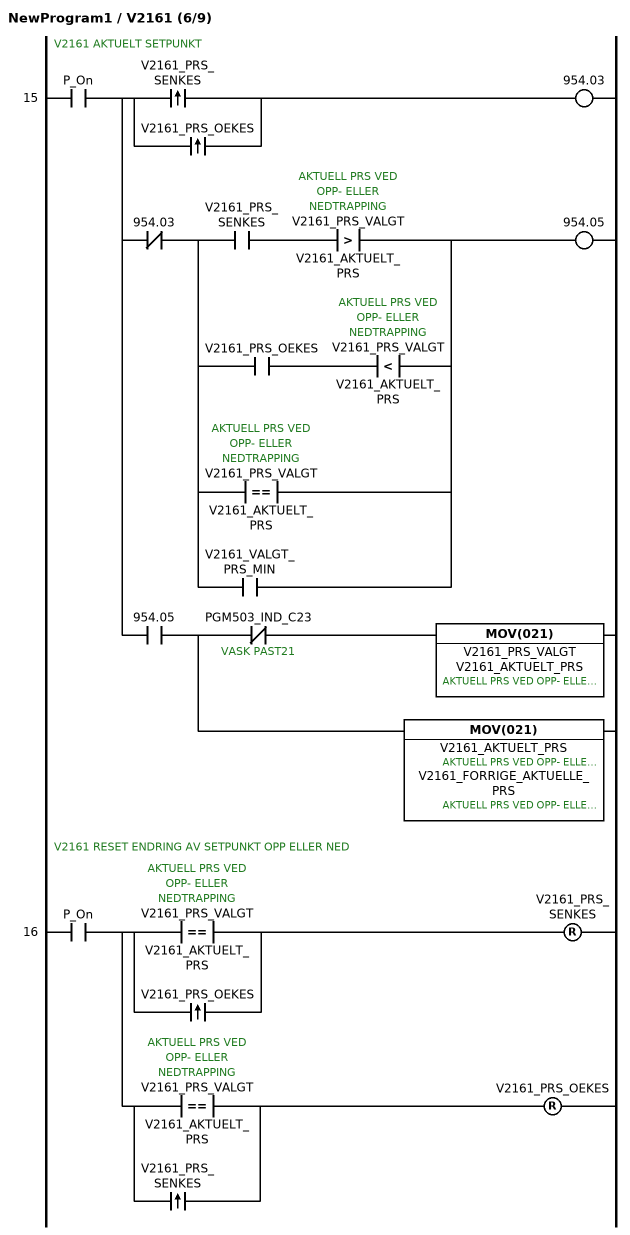
; [picture p1080: NewProgram1 / V2161, rungs 15-16]
; rung 15: V2161 AKTUELT SETPUNKT
LD P_On
OUT TR0
@LD V2161_PRS_SENKES
@OR V2161_PRS_OEKES
ANDLD
OUT 954.03
LD TR0
ANDNOT 954.03
LD V2161_PRS_SENKES
AND>(320) V2161_PRS_VALGT V2161_AKTUELT_PRS  ; AKTUELL PRS VED OPP- ELLER NEDTRAPPING
LD V2161_PRS_OEKES
AND<(310) V2161_PRS_VALGT V2161_AKTUELT_PRS  ; AKTUELL PRS VED OPP- ELLER NEDTRAPPING
ORLD
OR=(300) V2161_PRS_VALGT V2161_AKTUELT_PRS  ; AKTUELL PRS VED OPP- ELLER NEDTRAPPING
OR V2161_VALGT_PRS_MIN
ANDLD
OUT 954.05
LD TR0
AND 954.05
OUT TR0
ANDNOT PGM503_IND_C23  ; VASK PAST21
MOV(021) V2161_PRS_VALGT V2161_AKTUELT_PRS  ; AKTUELL PRS VED OPP- ELLER NEDTRAPPING
LD TR0
MOV(021) V2161_AKTUELT_PRS V2161_FORRIGE_AKTUELLE_PRS  ; AKTUELL PRS VED OPP- ELLER NEDTRAPPING
; rung 16: V2161 RESET ENDRING AV SETPUNKT OPP ELLER NED
LD P_On
OUT TR0
LD=(300) V2161_PRS_VALGT V2161_AKTUELT_PRS  ; AKTUELL PRS VED OPP- ELLER NEDTRAPPING
@OR V2161_PRS_OEKES
ANDLD
RSET V2161_PRS_SENKES
LD TR0
LD=(300) V2161_PRS_VALGT V2161_AKTUELT_PRS  ; AKTUELL PRS VED OPP- ELLER NEDTRAPPING
@OR V2161_PRS_SENKES
ANDLD
RSET V2161_PRS_OEKES

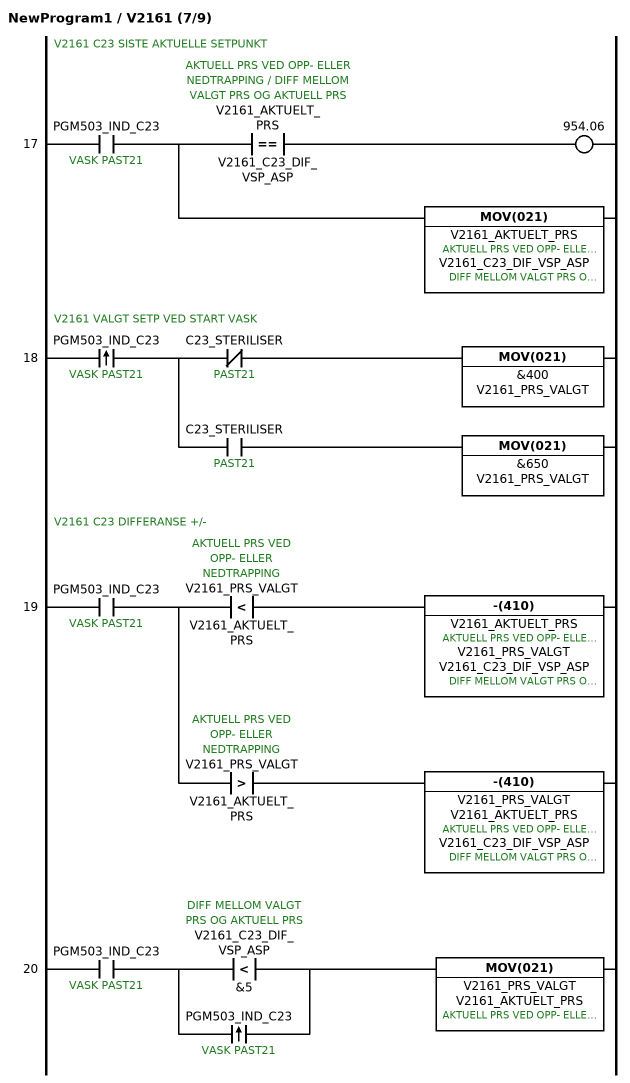
; rung 17: V2161 C23 SISTE AKTUELLE SETPUNKT
LD PGM503_IND_C23  ; VASK PAST21
OUT TR0
AND=(300) V2161_AKTUELT_PRS V2161_C23_DIF_VSP_ASP  ; AKTUELL PRS VED OPP- ELLER NEDTRAPPING, DIFF MELLOM VALGT PRS OG AKTUELL PRS
OUT 954.06
LD TR0
MOV(021) V2161_AKTUELT_PRS V2161_C23_DIF_VSP_ASP  ; AKTUELL PRS VED OPP- ELLER NEDTRAPPING, DIFF MELLOM VALGT PRS OG AKTUELL PRS
; rung 18: V2161 VALGT SETP VED START VASK
@LD PGM503_IND_C23  ; VASK PAST21
OUT TR0
ANDNOT C23_STERILISER  ; PAST21
MOV(021) &400 V2161_PRS_VALGT
LD TR0
AND C23_STERILISER  ; PAST21
MOV(021) &650 V2161_PRS_VALGT
; rung 19: V2161 C23 DIFFERANSE +/-
LD PGM503_IND_C23  ; VASK PAST21
OUT TR0
AND<(310) V2161_PRS_VALGT V2161_AKTUELT_PRS  ; AKTUELL PRS VED OPP- ELLER NEDTRAPPING
-(410) V2161_AKTUELT_PRS V2161_PRS_VALGT V2161_C23_DIF_VSP_ASP  ; AKTUELL PRS VED OPP- ELLER NEDTRAPPING, DIFF MELLOM VALGT PRS OG AKTUELL PRS
LD TR0
AND>(320) V2161_PRS_VALGT V2161_AKTUELT_PRS  ; AKTUELL PRS VED OPP- ELLER NEDTRAPPING
-(410) V2161_PRS_VALGT V2161_AKTUELT_PRS V2161_C23_DIF_VSP_ASP  ; AKTUELL PRS VED OPP- ELLER NEDTRAPPING, DIFF MELLOM VALGT PRS OG AKTUELL PRS
; rung 20
LD PGM503_IND_C23  ; VASK PAST21
LD<(310) V2161_C23_DIF_VSP_ASP &5  ; DIFF MELLOM VALGT PRS OG AKTUELL PRS
@OR PGM503_IND_C23  ; VASK PAST21
ANDLD
MOV(021) V2161_PRS_VALGT V2161_AKTUELT_PRS  ; AKTUELL PRS VED OPP- ELLER NEDTRAPPING

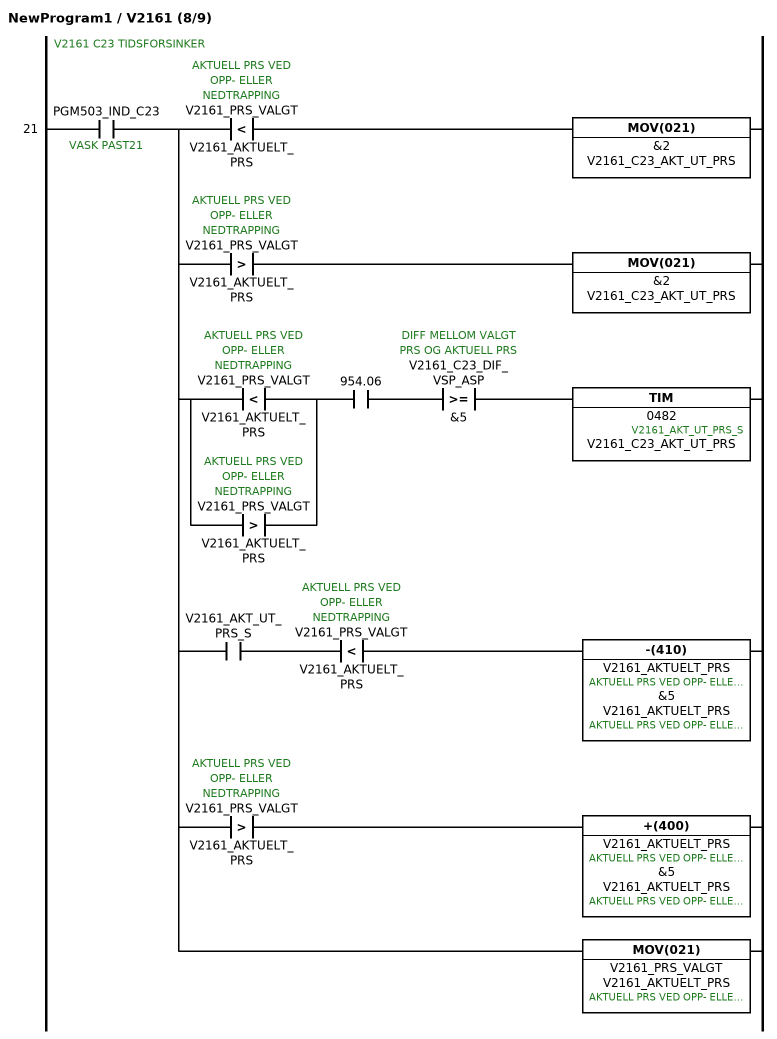
; rung 21: V2161 C23 TIDSFORSINKER
LD PGM503_IND_C23  ; VASK PAST21
OUT TR0
AND<(310) V2161_PRS_VALGT V2161_AKTUELT_PRS  ; AKTUELL PRS VED OPP- ELLER NEDTRAPPING
MOV(021) &2 V2161_C23_AKT_UT_PRS
LD TR0
AND>(320) V2161_PRS_VALGT V2161_AKTUELT_PRS  ; AKTUELL PRS VED OPP- ELLER NEDTRAPPING
MOV(021) &2 V2161_C23_AKT_UT_PRS
LD TR0
LD<(310) V2161_PRS_VALGT V2161_AKTUELT_PRS  ; AKTUELL PRS VED OPP- ELLER NEDTRAPPING
OR>(320) V2161_PRS_VALGT V2161_AKTUELT_PRS  ; AKTUELL PRS VED OPP- ELLER NEDTRAPPING
ANDLD
AND 954.06
AND>=(325) V2161_C23_DIF_VSP_ASP &5  ; DIFF MELLOM VALGT PRS OG AKTUELL PRS
TIM 0482 V2161_C23_AKT_UT_PRS  ; V2161_AKT_UT_PRS_S
LD TR0
AND V2161_AKT_UT_PRS_S
AND<(310) V2161_PRS_VALGT V2161_AKTUELT_PRS  ; AKTUELL PRS VED OPP- ELLER NEDTRAPPING
-(410) V2161_AKTUELT_PRS &5 V2161_AKTUELT_PRS  ; AKTUELL PRS VED OPP- ELLER NEDTRAPPING
LD TR0
AND>(320) V2161_PRS_VALGT V2161_AKTUELT_PRS  ; AKTUELL PRS VED OPP- ELLER NEDTRAPPING
+(400) V2161_AKTUELT_PRS &5 V2161_AKTUELT_PRS  ; AKTUELL PRS VED OPP- ELLER NEDTRAPPING
LD TR0
MOV(021) V2161_PRS_VALGT V2161_AKTUELT_PRS  ; AKTUELL PRS VED OPP- ELLER NEDTRAPPING

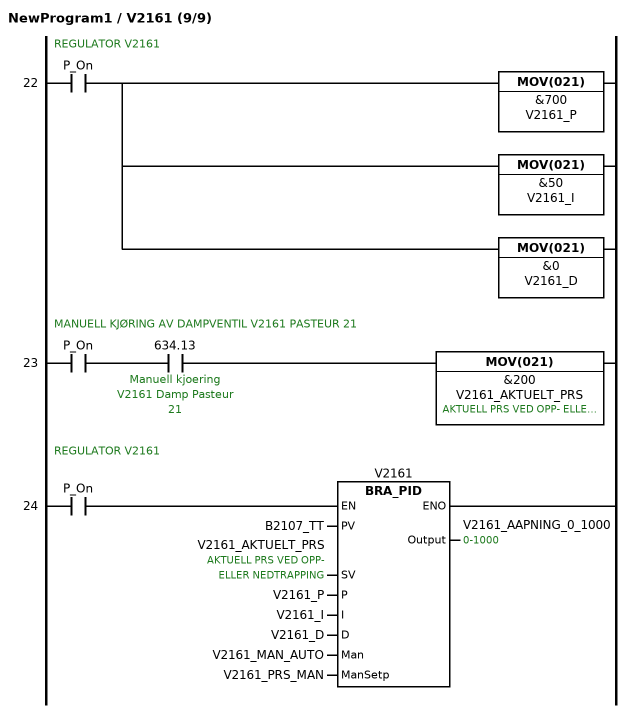
; rung 22: REGULATOR V2161
LD P_On
MOV(021) &700 V2161_P
MOV(021) &50 V2161_I
MOV(021) &0 V2161_D
; rung 23: MANUELL KJØRING AV DAMPVENTIL V2161 PASTEUR 21
LD P_On
AND 634.13  ; Manuell kjoering V2161 Damp Pasteur 21
MOV(021) &200 V2161_AKTUELT_PRS  ; AKTUELL PRS VED OPP- ELLER NEDTRAPPING
; rung 24: REGULATOR V2161
LD P_On
CALL V2161 : BRA_PID (PV := B2107_TT, SV := V2161_AKTUELT_PRS, P := V2161_P, I := V2161_I, D := V2161_D, Man := V2161_MAN_AUTO, ManSetp := V2161_PRS_MAN, Output => V2161_AAPNING_0_1000)  ; AKTUELL PRS VED OPP- ELLER NEDTRAPPING, 0-1000

### Section SEP21_KOMMUNIKASJ0N
; Kriterier: / - Separator går automatisk i "standby" etter "Start Up" / - Hvis ikke flow etter "Start Up", sett separator i "Feed Off" / - Ved skudd tar separator ikke mot nye kommandoer. La kommandoer stå høyt til ferdig. / GJENSTÅR: / - Kryssing av profibuss adresser

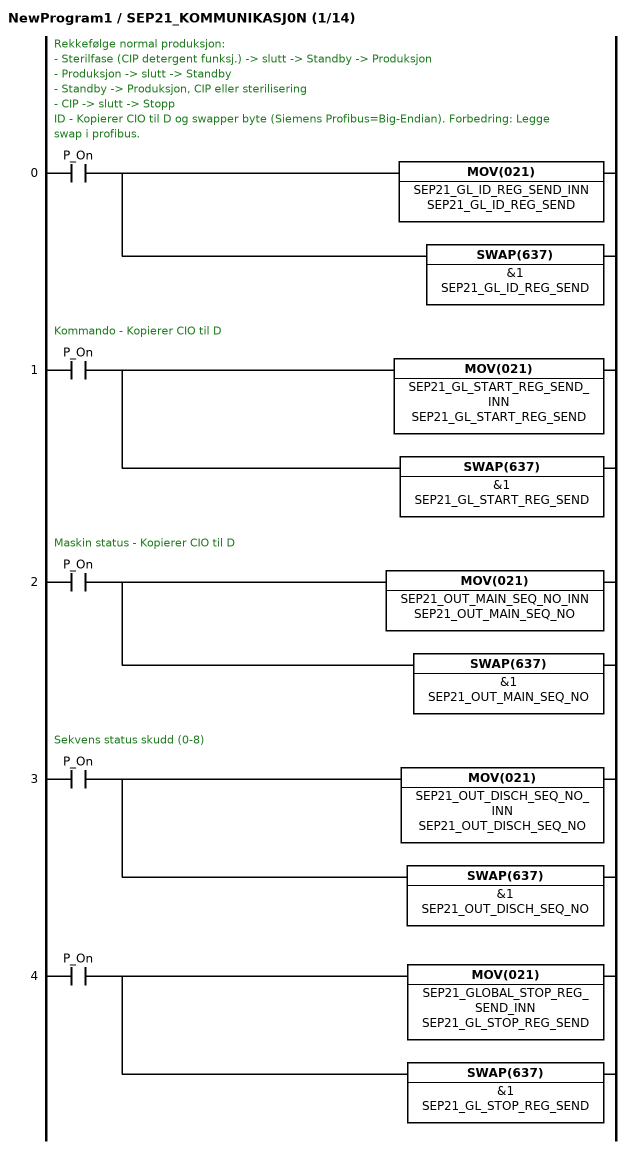
; rung 0: Rekkefølge normal produksjon: / - Sterilfase (CIP detergent funksj.) -> slutt -> Standby -> Produksjon / - Produksjon -> slutt -> Standby / - Standby -> Produksjon, CIP eller sterilisering / - CIP -> slutt -> Stopp / ID - Kopierer CIO til D og swapper byte (Siemens Profibus=Big-Endian). Forbedring: Legge swap i profibus.
LD P_On
MOV(021) SEP21_GL_ID_REG_SEND_INN SEP21_GL_ID_REG_SEND
SWAP(637) &1 SEP21_GL_ID_REG_SEND
; rung 1: Kommando - Kopierer CIO til D
LD P_On
MOV(021) SEP21_GL_START_REG_SEND_INN SEP21_GL_START_REG_SEND
SWAP(637) &1 SEP21_GL_START_REG_SEND
; rung 2: Maskin status - Kopierer CIO til D
LD P_On
MOV(021) SEP21_OUT_MAIN_SEQ_NO_INN SEP21_OUT_MAIN_SEQ_NO
SWAP(637) &1 SEP21_OUT_MAIN_SEQ_NO
; rung 3: Sekvens status skudd (0-8)
LD P_On
MOV(021) SEP21_OUT_DISCH_SEQ_NO_INN SEP21_OUT_DISCH_SEQ_NO
SWAP(637) &1 SEP21_OUT_DISCH_SEQ_NO
; rung 4
LD P_On
MOV(021) SEP21_GLOBAL_STOP_REG_SEND_INN SEP21_GL_STOP_REG_SEND
SWAP(637) &1 SEP21_GL_STOP_REG_SEND

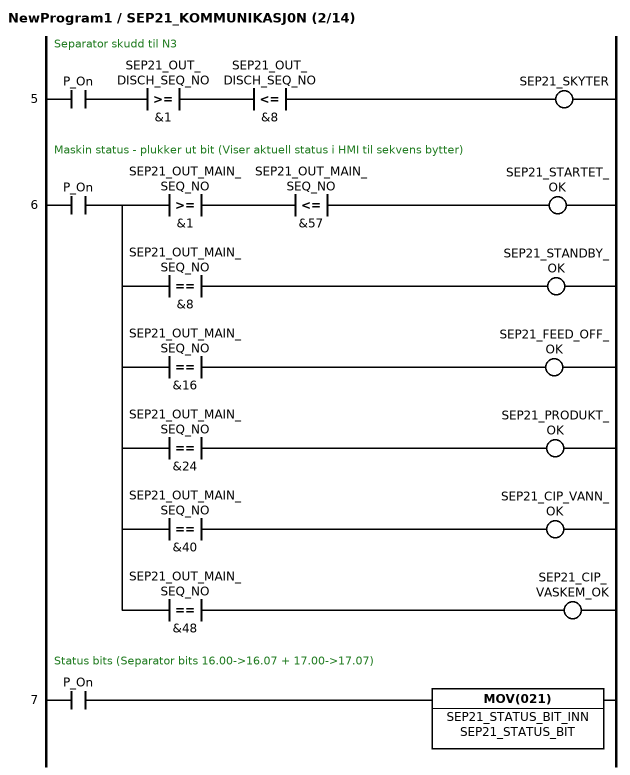
; rung 5: Separator skudd til N3
LD P_On
AND>=(325) SEP21_OUT_DISCH_SEQ_NO &1
AND<=(315) SEP21_OUT_DISCH_SEQ_NO &8
OUT SEP21_SKYTER
; rung 6: Maskin status - plukker ut bit (Viser aktuell status i HMI til sekvens bytter)
LD P_On
OUT TR0
AND>=(325) SEP21_OUT_MAIN_SEQ_NO &1
AND<=(315) SEP21_OUT_MAIN_SEQ_NO &57
OUT SEP21_STARTET_OK
LD TR0
AND=(300) SEP21_OUT_MAIN_SEQ_NO &8
OUT SEP21_STANDBY_OK
LD TR0
AND=(300) SEP21_OUT_MAIN_SEQ_NO &16
OUT SEP21_FEED_OFF_OK
LD TR0
AND=(300) SEP21_OUT_MAIN_SEQ_NO &24
OUT SEP21_PRODUKT_OK
LD TR0
AND=(300) SEP21_OUT_MAIN_SEQ_NO &40
OUT SEP21_CIP_VANN_OK
LD TR0
AND=(300) SEP21_OUT_MAIN_SEQ_NO &48
OUT SEP21_CIP_VASKEM_OK
; rung 7: Status bits (Separator bits 16.00->16.07 + 17.00->17.07)
LD P_On
MOV(021) SEP21_STATUS_BIT_INN SEP21_STATUS_BIT

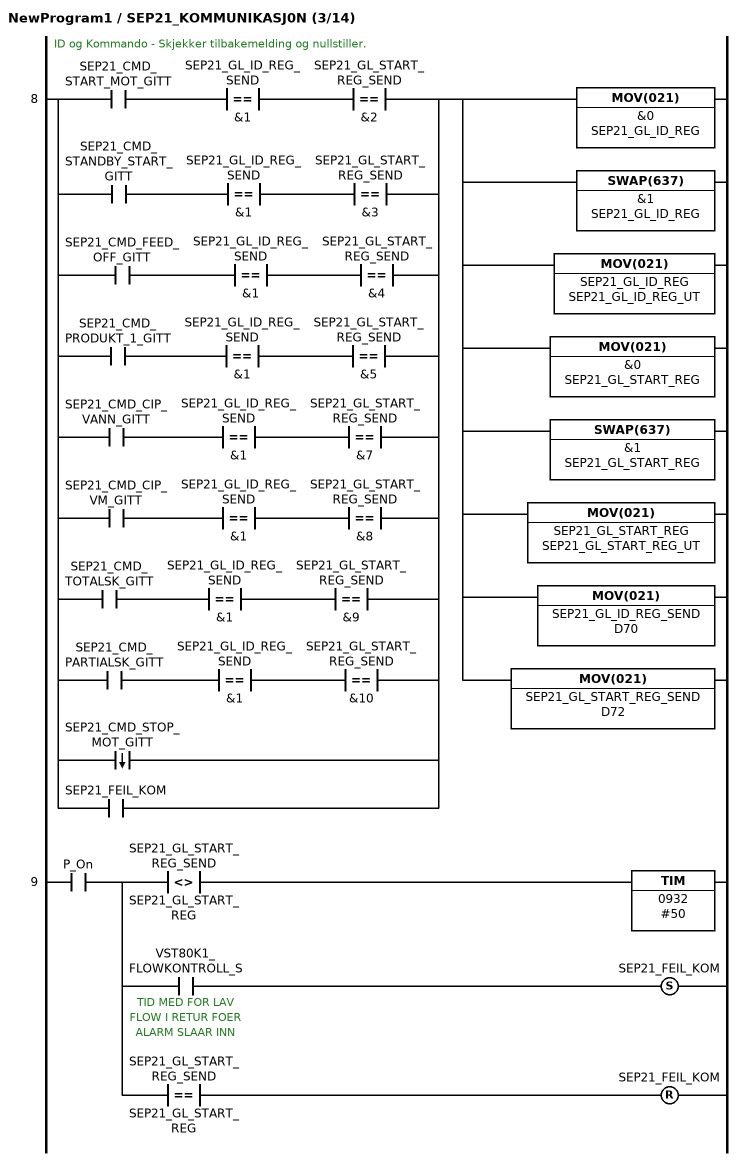
; rung 8: ID og Kommando - Skjekker tilbakemelding og nullstiller.
LD SEP21_CMD_START_MOT_GITT
AND=(300) SEP21_GL_ID_REG_SEND &1
AND=(300) SEP21_GL_START_REG_SEND &2
LD SEP21_CMD_STANDBY_START_GITT
AND=(300) SEP21_GL_ID_REG_SEND &1
AND=(300) SEP21_GL_START_REG_SEND &3
ORLD
LD SEP21_CMD_FEED_OFF_GITT
AND=(300) SEP21_GL_ID_REG_SEND &1
AND=(300) SEP21_GL_START_REG_SEND &4
ORLD
LD SEP21_CMD_PRODUKT_1_GITT
AND=(300) SEP21_GL_ID_REG_SEND &1
AND=(300) SEP21_GL_START_REG_SEND &5
ORLD
LD SEP21_CMD_CIP_VANN_GITT
AND=(300) SEP21_GL_ID_REG_SEND &1
AND=(300) SEP21_GL_START_REG_SEND &7
ORLD
LD SEP21_CMD_CIP_VM_GITT
AND=(300) SEP21_GL_ID_REG_SEND &1
AND=(300) SEP21_GL_START_REG_SEND &8
ORLD
LD SEP21_CMD_TOTALSK_GITT
AND=(300) SEP21_GL_ID_REG_SEND &1
AND=(300) SEP21_GL_START_REG_SEND &9
ORLD
LD SEP21_CMD_PARTIALSK_GITT
AND=(300) SEP21_GL_ID_REG_SEND &1
AND=(300) SEP21_GL_START_REG_SEND &10
ORLD
%OR SEP21_CMD_STOP_MOT_GITT  // Hvis stop så nullstill register
OR SEP21_FEIL_KOM
MOV(021) &0 SEP21_GL_ID_REG
SWAP(637) &1 SEP21_GL_ID_REG
MOV(021) SEP21_GL_ID_REG SEP21_GL_ID_REG_UT
MOV(021) &0 SEP21_GL_START_REG
SWAP(637) &1 SEP21_GL_START_REG
MOV(021) SEP21_GL_START_REG SEP21_GL_START_REG_UT
MOV(021) SEP21_GL_ID_REG_SEND D70  // For test - Siste ID som er mottatt
MOV(021) SEP21_GL_START_REG_SEND D72  // For test - Siste KOMMANDO som er mottatt
; rung 9
LD P_On
OUT TR0
AND<>(305) SEP21_GL_START_REG_SEND SEP21_GL_START_REG
TIM 0932 #50
LD TR0
AND VST80K1_FLOWKONTROLL_S  ; TID MED FOR LAV FLOW I RETUR FOER ALARM SLAAR INN
SET SEP21_FEIL_KOM
LD TR0
AND=(300) SEP21_GL_START_REG_SEND SEP21_GL_START_REG
RSET SEP21_FEIL_KOM

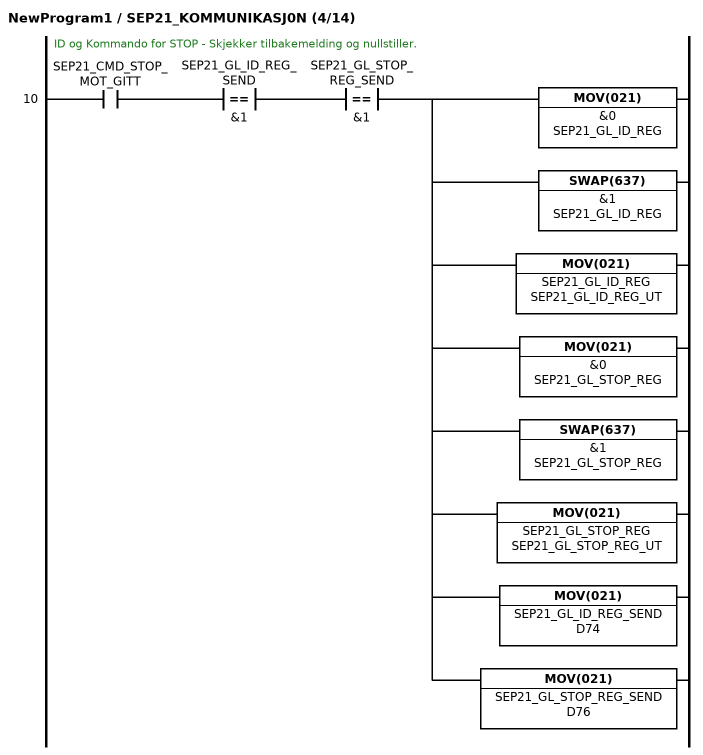
; rung 10: ID og Kommando for STOP - Skjekker tilbakemelding og nullstiller.
LD SEP21_CMD_STOP_MOT_GITT
AND=(300) SEP21_GL_ID_REG_SEND &1
AND=(300) SEP21_GL_STOP_REG_SEND &1
MOV(021) &0 SEP21_GL_ID_REG
SWAP(637) &1 SEP21_GL_ID_REG
MOV(021) SEP21_GL_ID_REG SEP21_GL_ID_REG_UT
MOV(021) &0 SEP21_GL_STOP_REG
SWAP(637) &1 SEP21_GL_STOP_REG
MOV(021) SEP21_GL_STOP_REG SEP21_GL_STOP_REG_UT
MOV(021) SEP21_GL_ID_REG_SEND D74  // For test - Siste STOP ID som er mottatt
MOV(021) SEP21_GL_STOP_REG_SEND D76  // For test - Siste STOP KOMMANDO som er mottatt

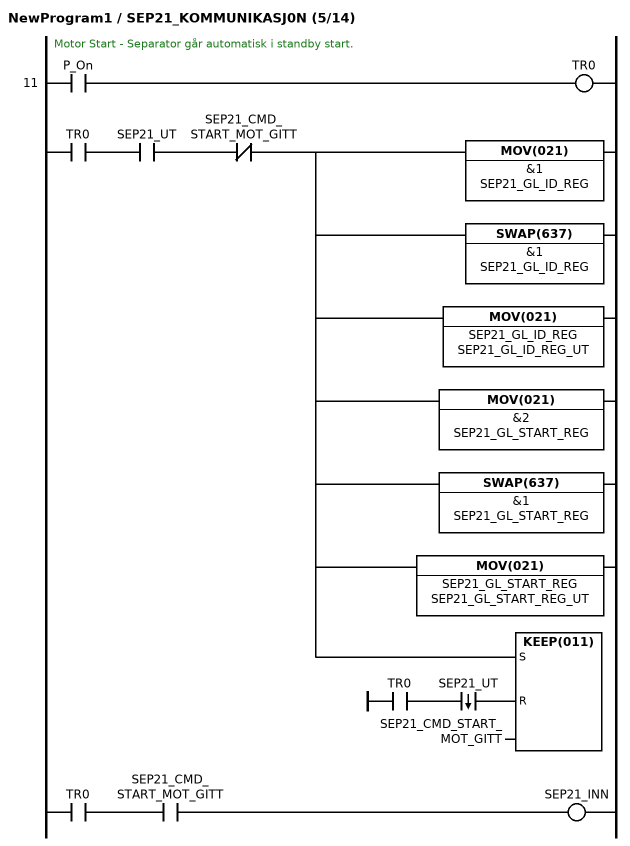
; rung 11: Motor Start - Separator går automatisk i standby start.
LD P_On
OUT TR0
AND SEP21_UT
ANDNOT SEP21_CMD_START_MOT_GITT
MOV(021) &1 SEP21_GL_ID_REG
SWAP(637) &1 SEP21_GL_ID_REG
MOV(021) SEP21_GL_ID_REG SEP21_GL_ID_REG_UT
MOV(021) &2 SEP21_GL_START_REG
SWAP(637) &1 SEP21_GL_START_REG
MOV(021) SEP21_GL_START_REG SEP21_GL_START_REG_UT
LD TR0
%AND SEP21_UT
KEEP(011) SEP21_CMD_START_MOT_GITT
LD TR0
AND SEP21_CMD_START_MOT_GITT
OUT SEP21_INN

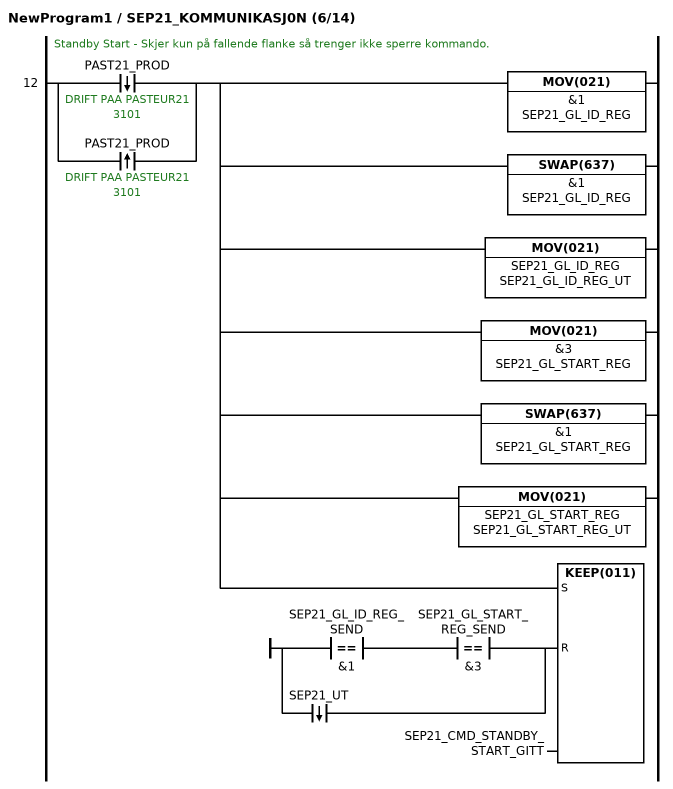
; rung 12: Standby Start - Skjer kun på fallende flanke så trenger ikke sperre kommando.
%LD PAST21_PROD  ; DRIFT PAA PASTEUR21 3101
@OR PAST21_PROD  ; DRIFT PAA PASTEUR21 3101  // Kan ikke gå direkte til prod 1 fra CIP detergent. Må via Standby, stopp eller CIP vann.
MOV(021) &1 SEP21_GL_ID_REG
SWAP(637) &1 SEP21_GL_ID_REG
MOV(021) SEP21_GL_ID_REG SEP21_GL_ID_REG_UT
MOV(021) &3 SEP21_GL_START_REG
SWAP(637) &1 SEP21_GL_START_REG
MOV(021) SEP21_GL_START_REG SEP21_GL_START_REG_UT
LD=(300) SEP21_GL_ID_REG_SEND &1
AND=(300) SEP21_GL_START_REG_SEND &3
%OR SEP21_UT
KEEP(011) SEP21_CMD_STANDBY_START_GITT

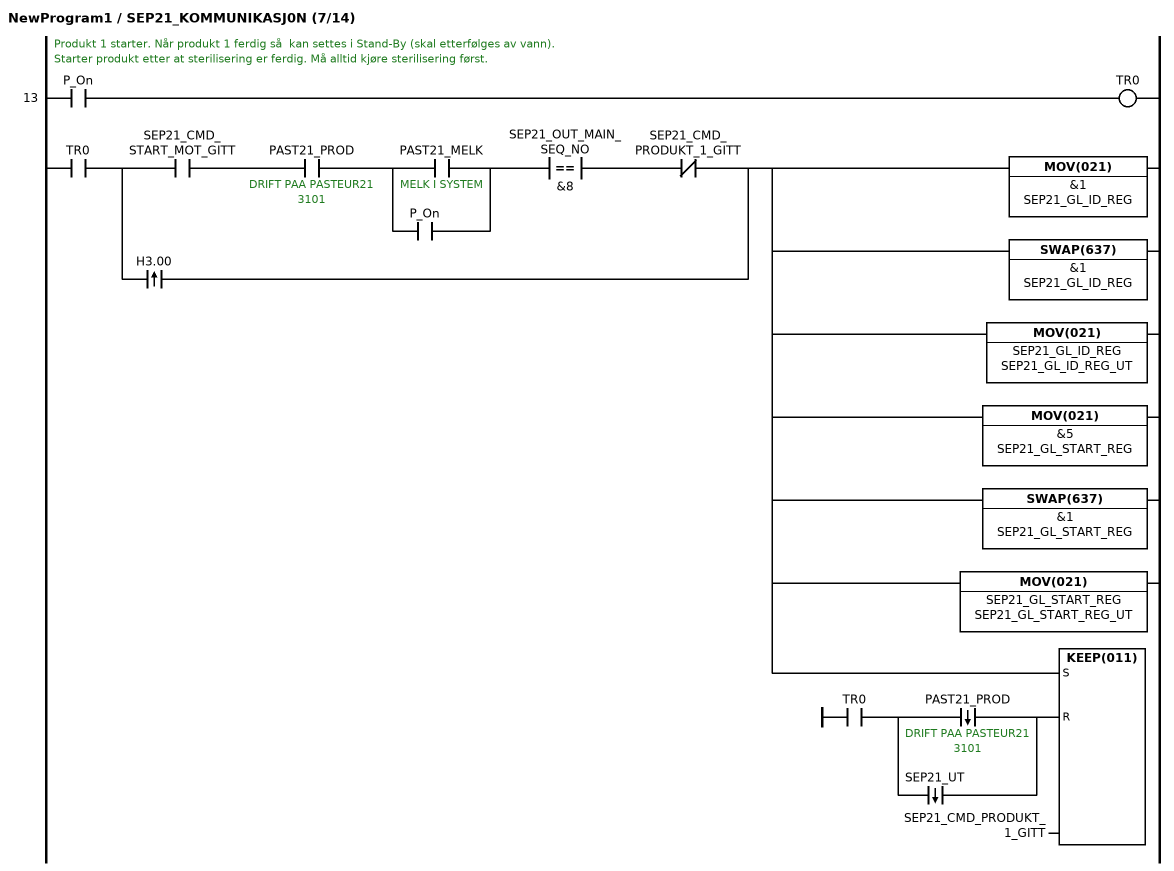
; rung 13: Produkt 1 starter. Når produkt 1 ferdig så  kan settes i Stand-By (skal etterfølges av vann). / Starter produkt etter at sterilisering er ferdig. Må alltid kjøre sterilisering først.
LD P_On
OUT TR0
LD SEP21_CMD_START_MOT_GITT
AND PAST21_PROD  ; DRIFT PAA PASTEUR21 3101
LD PAST21_MELK  ; MELK I SYSTEM
OR P_On
ANDLD
AND=(300) SEP21_OUT_MAIN_SEQ_NO &8  // Kann ikke gå direkte til prod1 fra CIP detergent (se manual). Må via Standby.
ANDNOT SEP21_CMD_PRODUKT_1_GITT
@OR H3.00
ANDLD
MOV(021) &1 SEP21_GL_ID_REG
SWAP(637) &1 SEP21_GL_ID_REG
MOV(021) SEP21_GL_ID_REG SEP21_GL_ID_REG_UT
MOV(021) &5 SEP21_GL_START_REG
SWAP(637) &1 SEP21_GL_START_REG
MOV(021) SEP21_GL_START_REG SEP21_GL_START_REG_UT
LD TR0
%LD PAST21_PROD  ; DRIFT PAA PASTEUR21 3101
%OR SEP21_UT
ANDLD
KEEP(011) SEP21_CMD_PRODUKT_1_GITT

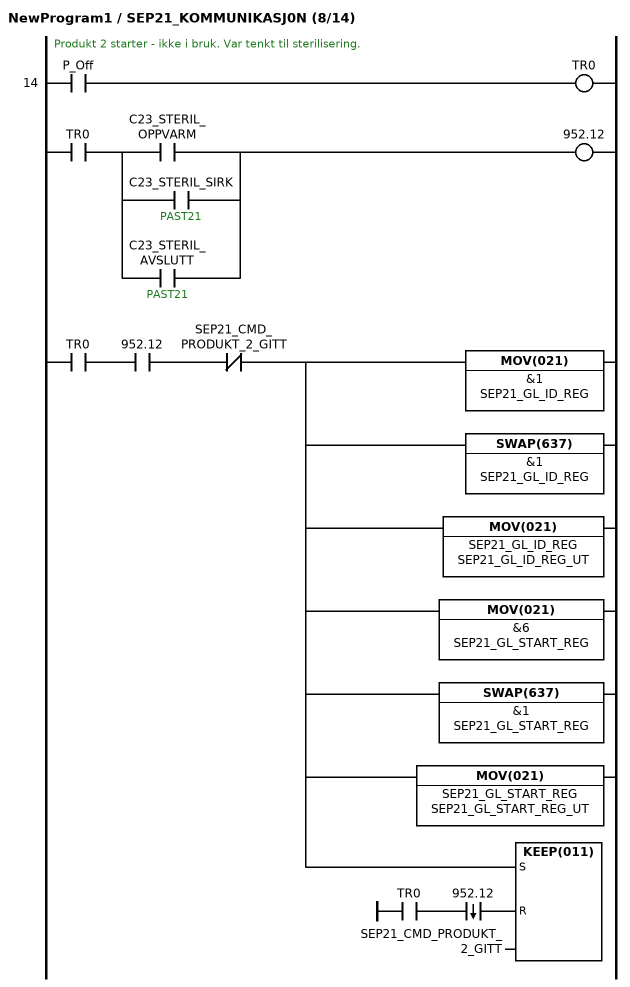
; rung 14: Produkt 2 starter - ikke i bruk. Var tenkt til sterilisering.
LD P_Off
OUT TR0
LD C23_STERIL_OPPVARM
OR C23_STERIL_SIRK  ; PAST21
OR C23_STERIL_AVSLUTT  ; PAST21
ANDLD
OUT 952.12
LD TR0
AND 952.12
ANDNOT SEP21_CMD_PRODUKT_2_GITT
MOV(021) &1 SEP21_GL_ID_REG
SWAP(637) &1 SEP21_GL_ID_REG
MOV(021) SEP21_GL_ID_REG SEP21_GL_ID_REG_UT
MOV(021) &6 SEP21_GL_START_REG
SWAP(637) &1 SEP21_GL_START_REG
MOV(021) SEP21_GL_START_REG SEP21_GL_START_REG_UT
LD TR0
%AND 952.12
KEEP(011) SEP21_CMD_PRODUKT_2_GITT

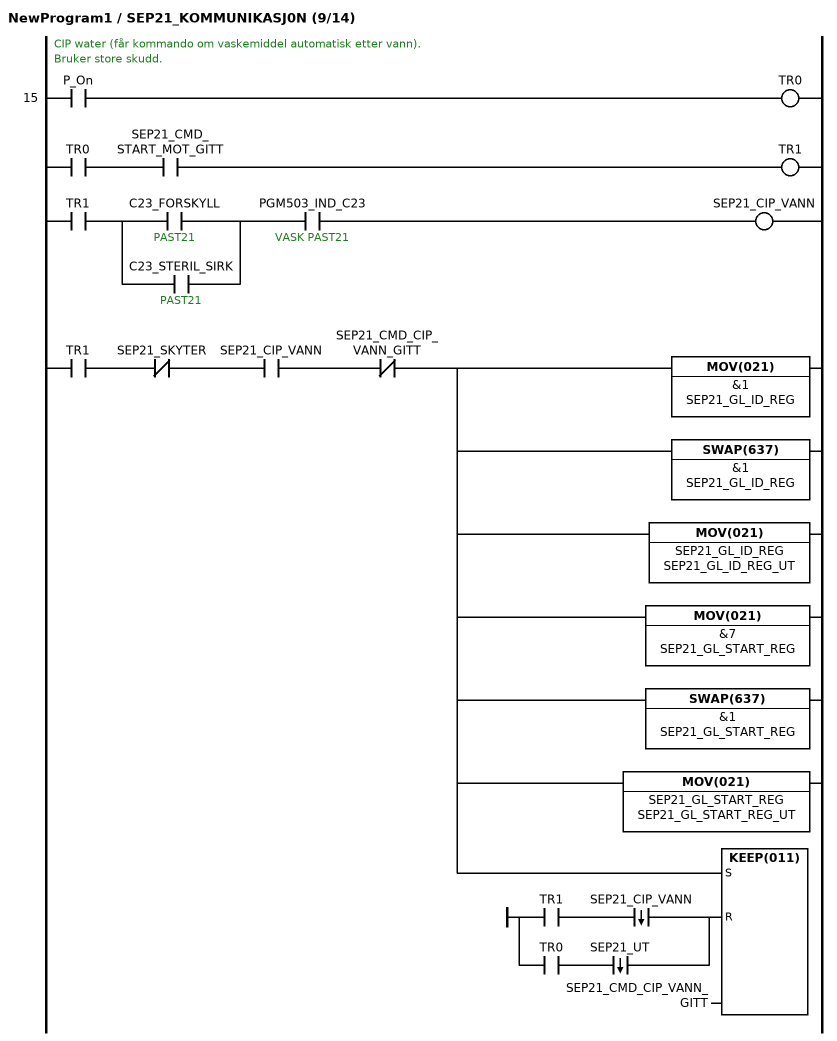
; rung 15: CIP water (får kommando om vaskemiddel automatisk etter vann). / Bruker store skudd.
LD P_On
OUT TR0
AND SEP21_CMD_START_MOT_GITT
OUT TR1
LD C23_FORSKYLL  ; PAST21
OR C23_STERIL_SIRK  ; PAST21
ANDLD
AND PGM503_IND_C23  ; VASK PAST21
OUT SEP21_CIP_VANN
LD TR1
ANDNOT SEP21_SKYTER
AND SEP21_CIP_VANN
ANDNOT SEP21_CMD_CIP_VANN_GITT
MOV(021) &1 SEP21_GL_ID_REG
SWAP(637) &1 SEP21_GL_ID_REG
MOV(021) SEP21_GL_ID_REG SEP21_GL_ID_REG_UT
MOV(021) &7 SEP21_GL_START_REG
SWAP(637) &1 SEP21_GL_START_REG
MOV(021) SEP21_GL_START_REG SEP21_GL_START_REG_UT
LD TR1
%AND SEP21_CIP_VANN
LD TR0
%AND SEP21_UT
ORLD
KEEP(011) SEP21_CMD_CIP_VANN_GITT

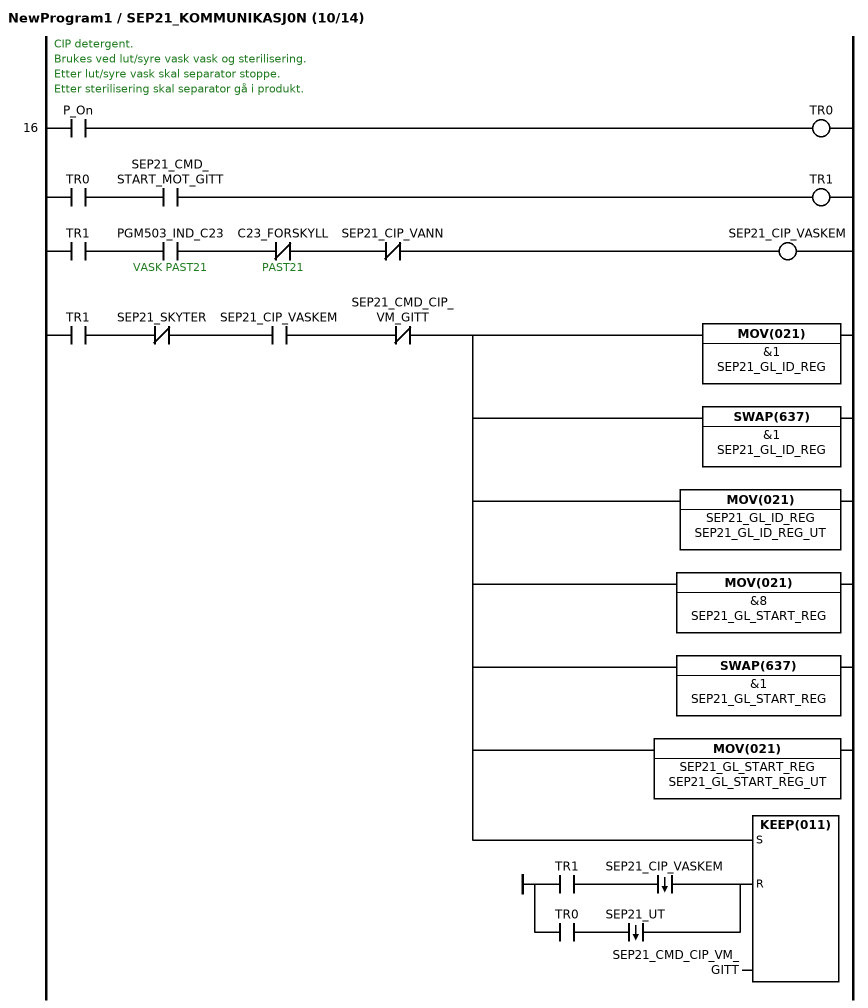
; rung 16: CIP detergent. / Brukes ved lut/syre vask vask og sterilisering. / Etter lut/syre vask skal separator stoppe. / Etter sterilisering skal separator gå i produkt.
LD P_On
OUT TR0
AND SEP21_CMD_START_MOT_GITT
OUT TR1
AND PGM503_IND_C23  ; VASK PAST21
ANDNOT C23_FORSKYLL  ; PAST21
ANDNOT SEP21_CIP_VANN  // Midlertidig. 3616.11 toggler av/på ved start av CIP vann! Må rettes i Node3. / 3616.11 går også på ved sterilvask. Da trenger vi egentlig ikke sterilvask fra ipc så lenge CIP detergant kan brukes som sterilvask.
OUT SEP21_CIP_VASKEM
LD TR1
ANDNOT SEP21_SKYTER
AND SEP21_CIP_VASKEM
ANDNOT SEP21_CMD_CIP_VM_GITT
MOV(021) &1 SEP21_GL_ID_REG
SWAP(637) &1 SEP21_GL_ID_REG
MOV(021) SEP21_GL_ID_REG SEP21_GL_ID_REG_UT
MOV(021) &8 SEP21_GL_START_REG
SWAP(637) &1 SEP21_GL_START_REG
MOV(021) SEP21_GL_START_REG SEP21_GL_START_REG_UT
LD TR1
%AND SEP21_CIP_VASKEM
LD TR0
%AND SEP21_UT
ORLD
KEEP(011) SEP21_CMD_CIP_VM_GITT

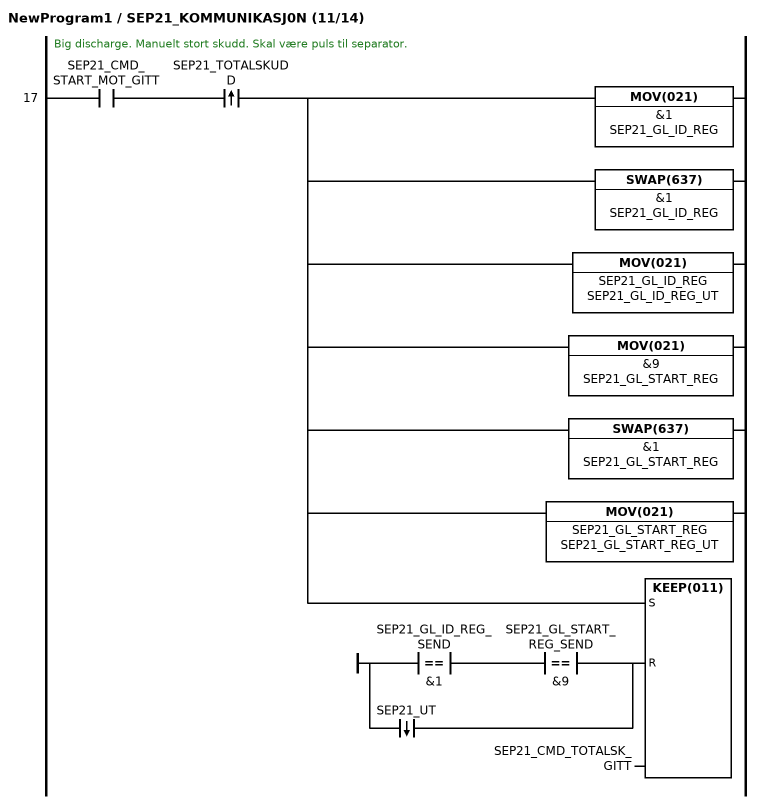
; rung 17: Big discharge. Manuelt stort skudd. Skal være puls til separator.
LD SEP21_CMD_START_MOT_GITT
@AND SEP21_TOTALSKUDD
MOV(021) &1 SEP21_GL_ID_REG
SWAP(637) &1 SEP21_GL_ID_REG
MOV(021) SEP21_GL_ID_REG SEP21_GL_ID_REG_UT
MOV(021) &9 SEP21_GL_START_REG
SWAP(637) &1 SEP21_GL_START_REG
MOV(021) SEP21_GL_START_REG SEP21_GL_START_REG_UT
LD=(300) SEP21_GL_ID_REG_SEND &1
AND=(300) SEP21_GL_START_REG_SEND &9
%OR SEP21_UT
KEEP(011) SEP21_CMD_TOTALSK_GITT

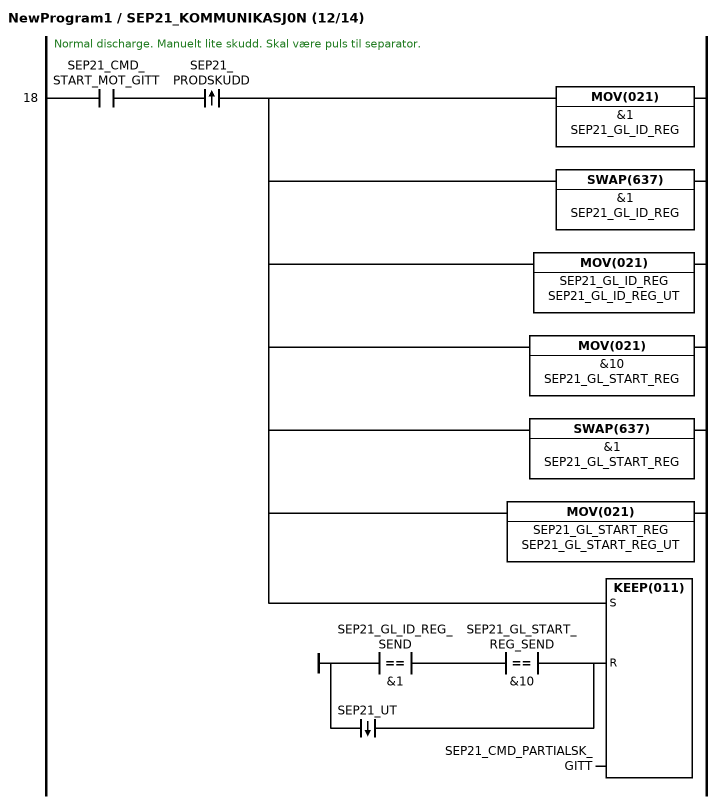
; rung 18: Normal discharge. Manuelt lite skudd. Skal være puls til separator.
LD SEP21_CMD_START_MOT_GITT
@AND SEP21_PRODSKUDD
MOV(021) &1 SEP21_GL_ID_REG
SWAP(637) &1 SEP21_GL_ID_REG
MOV(021) SEP21_GL_ID_REG SEP21_GL_ID_REG_UT
MOV(021) &10 SEP21_GL_START_REG
SWAP(637) &1 SEP21_GL_START_REG
MOV(021) SEP21_GL_START_REG SEP21_GL_START_REG_UT
LD=(300) SEP21_GL_ID_REG_SEND &1
AND=(300) SEP21_GL_START_REG_SEND &10
%OR SEP21_UT
KEEP(011) SEP21_CMD_PARTIALSK_GITT

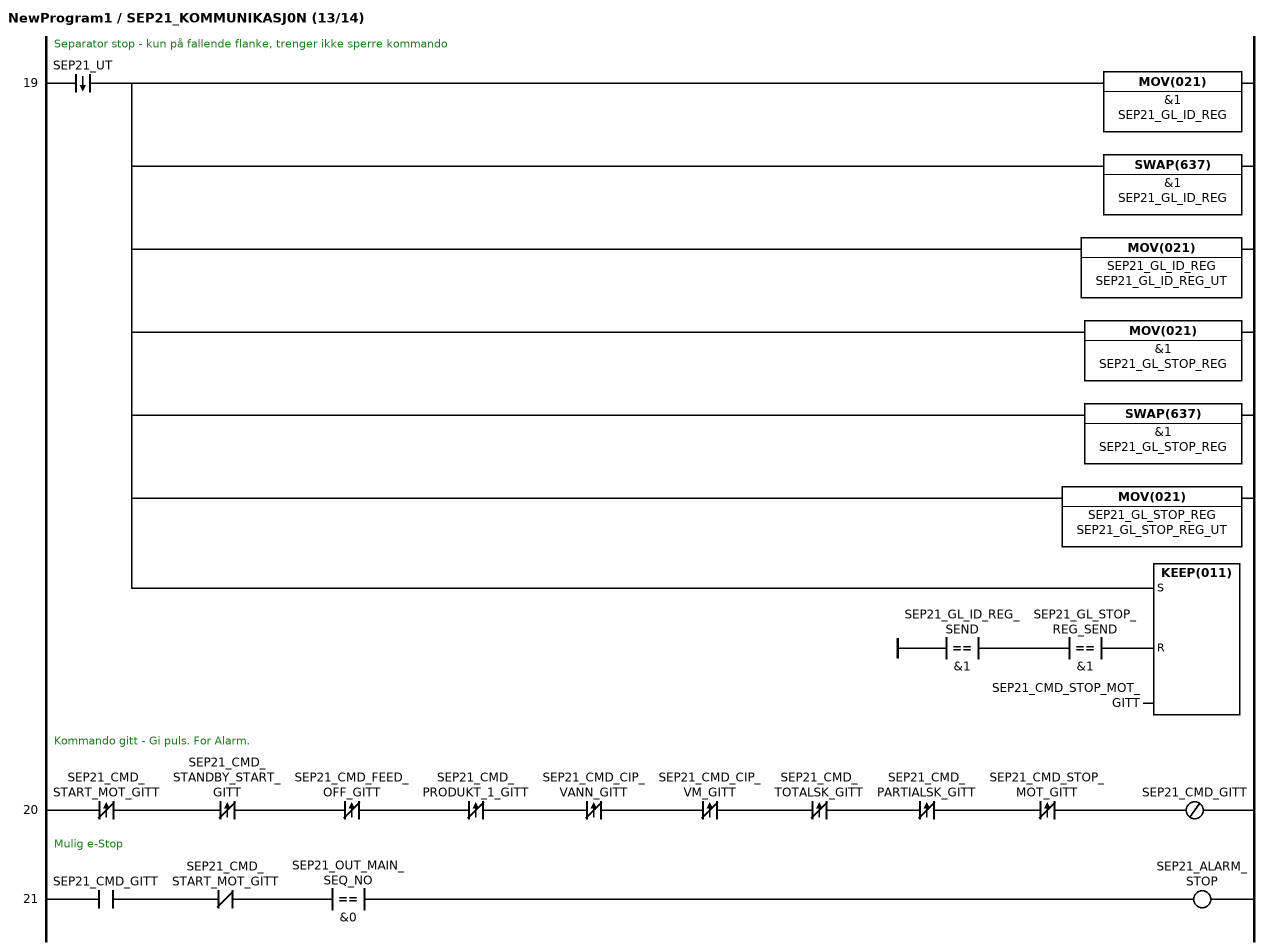
; rung 19: Separator stop - kun på fallende flanke, trenger ikke sperre kommando
%LD SEP21_UT
MOV(021) &1 SEP21_GL_ID_REG
SWAP(637) &1 SEP21_GL_ID_REG
MOV(021) SEP21_GL_ID_REG SEP21_GL_ID_REG_UT
MOV(021) &1 SEP21_GL_STOP_REG
SWAP(637) &1 SEP21_GL_STOP_REG
MOV(021) SEP21_GL_STOP_REG SEP21_GL_STOP_REG_UT
LD=(300) SEP21_GL_ID_REG_SEND &1
AND=(300) SEP21_GL_STOP_REG_SEND &1
KEEP(011) SEP21_CMD_STOP_MOT_GITT
; rung 20: Kommando gitt - Gi puls. For Alarm.
@LDNOT SEP21_CMD_START_MOT_GITT
@ANDNOT SEP21_CMD_STANDBY_START_GITT
@ANDNOT SEP21_CMD_FEED_OFF_GITT
@ANDNOT SEP21_CMD_PRODUKT_1_GITT
@ANDNOT SEP21_CMD_CIP_VANN_GITT
@ANDNOT SEP21_CMD_CIP_VM_GITT
@ANDNOT SEP21_CMD_TOTALSK_GITT
@ANDNOT SEP21_CMD_PARTIALSK_GITT
@ANDNOT SEP21_CMD_STOP_MOT_GITT
OUTNOT SEP21_CMD_GITT
; rung 21: Mulig e-Stop
LD SEP21_CMD_GITT
ANDNOT SEP21_CMD_START_MOT_GITT
AND=(300) SEP21_OUT_MAIN_SEQ_NO &0
OUT SEP21_ALARM_STOP

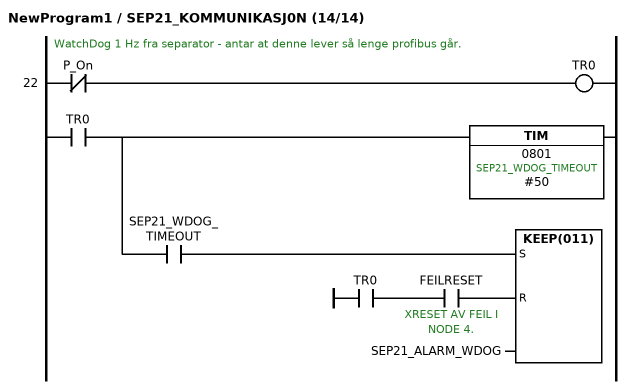
; rung 22: WatchDog 1 Hz fra separator - antar at denne lever så lenge profibus går.
LDNOT P_On
OUT TR0
TIM 0801 #50  ; SEP21_WDOG_TIMEOUT
AND SEP21_WDOG_TIMEOUT
LD TR0
AND FEILRESET  ; XRESET AV FEIL I NODE 4.
KEEP(011) SEP21_ALARM_WDOG

### Section SEP21_DRIFT

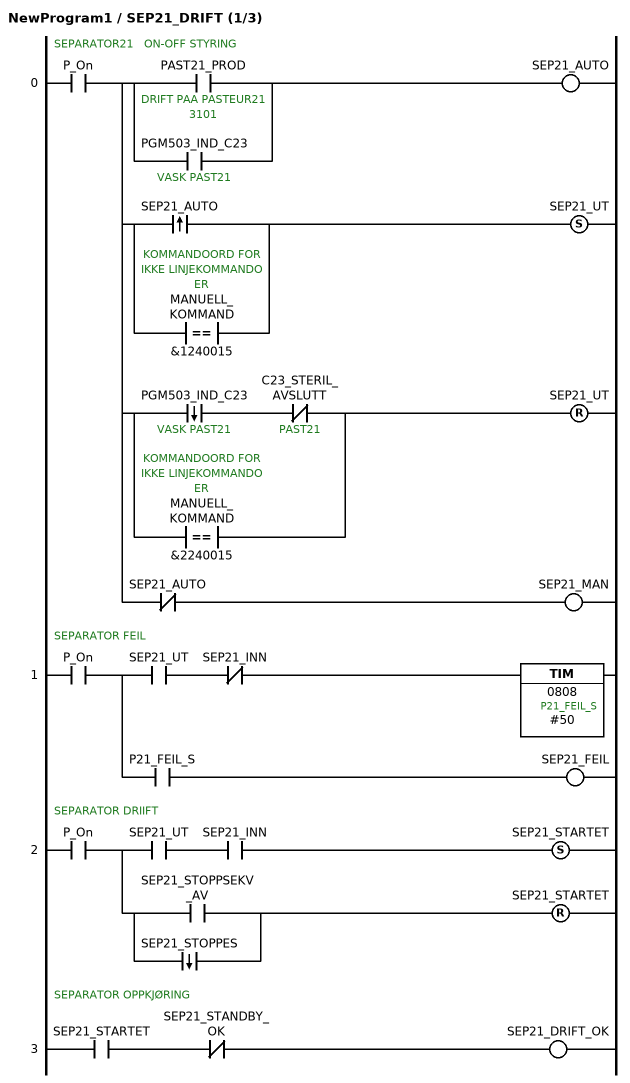
; rung 0: SEPARATOR21   ON-OFF STYRING
LD P_On
OUT TR0
LD PAST21_PROD  ; DRIFT PAA PASTEUR21 3101
OR PGM503_IND_C23  ; VASK PAST21
ANDLD
OUT SEP21_AUTO
LD TR0
@LD SEP21_AUTO
OR=L(301) MANUELL_KOMMAND &1240015  ; KOMMANDOORD FOR IKKE LINJEKOMMANDOER
ANDLD
SET SEP21_UT
LD TR0
%LD PGM503_IND_C23  ; VASK PAST21
ANDNOT C23_STERIL_AVSLUTT  ; PAST21
OR=L(301) MANUELL_KOMMAND &2240015  ; KOMMANDOORD FOR IKKE LINJEKOMMANDOER
ANDLD
RSET SEP21_UT
LD TR0
ANDNOT SEP21_AUTO
OUT SEP21_MAN
; rung 1: SEPARATOR FEIL
LD P_On
OUT TR0
AND SEP21_UT
ANDNOT SEP21_INN
TIM 0808 #50  ; P21_FEIL_S
LD TR0
AND P21_FEIL_S
OUT SEP21_FEIL
; rung 2: SEPARATOR DRIIFT
LD P_On
OUT TR0
AND SEP21_UT
AND SEP21_INN
SET SEP21_STARTET
LD TR0
LD SEP21_STOPPSEKV_AV
%OR SEP21_STOPPES
ANDLD
RSET SEP21_STARTET
; rung 3: SEPARATOR OPPKJØRING
LD SEP21_STARTET
ANDNOT SEP21_STANDBY_OK
OUT SEP21_DRIFT_OK

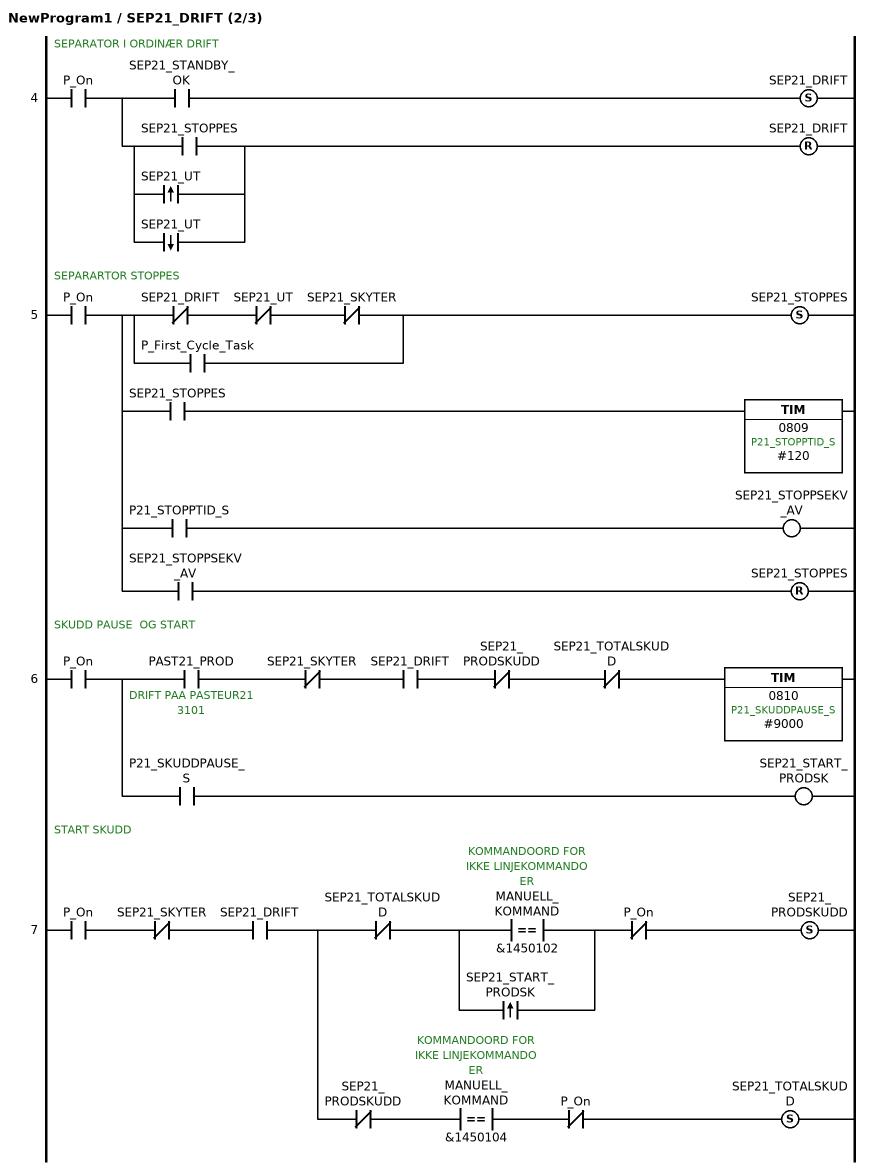
; rung 4: SEPARATOR I ORDINÆR DRIFT
LD P_On
OUT TR0
AND SEP21_STANDBY_OK
SET SEP21_DRIFT
LD TR0
LD SEP21_STOPPES
@OR SEP21_UT
%OR SEP21_UT
ANDLD
RSET SEP21_DRIFT
; rung 5: SEPARARTOR STOPPES
LD P_On
OUT TR0
LDNOT SEP21_DRIFT
ANDNOT SEP21_UT
ANDNOT SEP21_SKYTER
OR P_First_Cycle_Task
ANDLD
SET SEP21_STOPPES
LD TR0
AND SEP21_STOPPES
TIM 0809 #120  ; P21_STOPPTID_S
LD TR0
AND P21_STOPPTID_S
OUT SEP21_STOPPSEKV_AV
LD TR0
AND SEP21_STOPPSEKV_AV
RSET SEP21_STOPPES
; rung 6: SKUDD PAUSE  OG START
LD P_On
OUT TR0
AND PAST21_PROD  ; DRIFT PAA PASTEUR21 3101
ANDNOT SEP21_SKYTER
AND SEP21_DRIFT
ANDNOT SEP21_PRODSKUDD
ANDNOT SEP21_TOTALSKUDD
TIM 0810 #9000  ; P21_SKUDDPAUSE_S
LD TR0
AND P21_SKUDDPAUSE_S
OUT SEP21_START_PRODSK
; rung 7: START SKUDD
LD P_On
ANDNOT SEP21_SKYTER
AND SEP21_DRIFT
OUT TR0
ANDNOT SEP21_TOTALSKUDD
LD=L(301) MANUELL_KOMMAND &1450102  ; KOMMANDOORD FOR IKKE LINJEKOMMANDOER
@OR SEP21_START_PRODSK
ANDLD
ANDNOT P_On
SET SEP21_PRODSKUDD
LD TR0
ANDNOT SEP21_PRODSKUDD
AND=L(301) MANUELL_KOMMAND &1450104  ; KOMMANDOORD FOR IKKE LINJEKOMMANDOER
ANDNOT P_On
SET SEP21_TOTALSKUDD

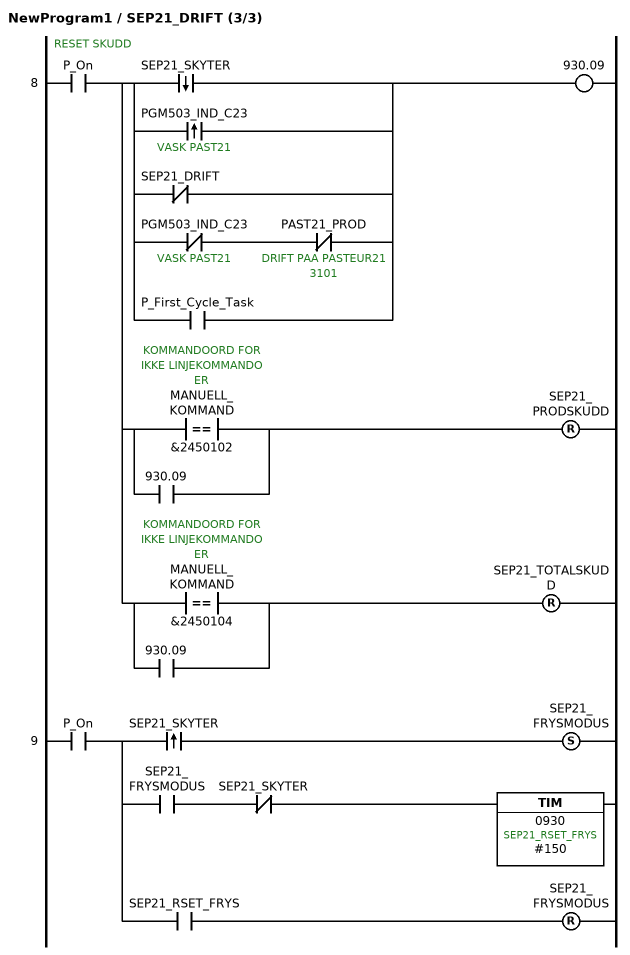
; rung 8: RESET SKUDD
LD P_On
OUT TR0
%LD SEP21_SKYTER
@OR PGM503_IND_C23  ; VASK PAST21
ORNOT SEP21_DRIFT
LDNOT PGM503_IND_C23  ; VASK PAST21
ANDNOT PAST21_PROD  ; DRIFT PAA PASTEUR21 3101
ORLD
OR P_First_Cycle_Task
ANDLD
OUT 930.09
LD TR0
LD=L(301) MANUELL_KOMMAND &2450102  ; KOMMANDOORD FOR IKKE LINJEKOMMANDOER
OR 930.09
ANDLD
RSET SEP21_PRODSKUDD
LD TR0
LD=L(301) MANUELL_KOMMAND &2450104  ; KOMMANDOORD FOR IKKE LINJEKOMMANDOER
OR 930.09
ANDLD
RSET SEP21_TOTALSKUDD
; rung 9
LD P_On
OUT TR0
@AND SEP21_SKYTER
SET SEP21_FRYSMODUS
LD TR0
AND SEP21_FRYSMODUS
ANDNOT SEP21_SKYTER
TIM 0930 #150  ; SEP21_RSET_FRYS
LD TR0
AND SEP21_RSET_FRYS
RSET SEP21_FRYSMODUS

### Section PAST_21_VENTILER

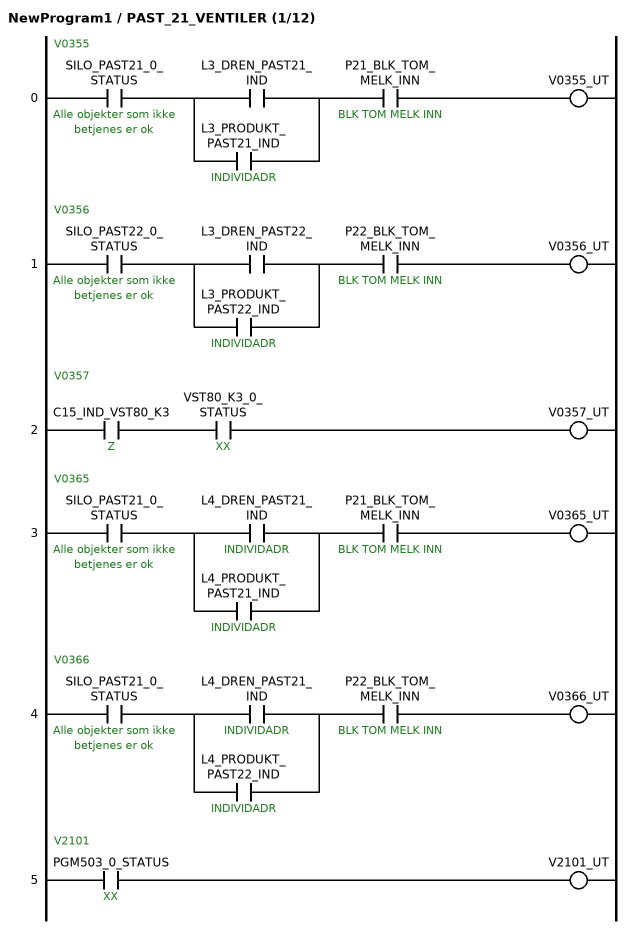
; rung 0: V0355
LD SILO_PAST21_0_STATUS  ; Alle objekter som ikke betjenes er ok
LD L3_DREN_PAST21_IND
OR L3_PRODUKT_PAST21_IND  ; INDIVIDADR
ANDLD
AND P21_BLK_TOM_MELK_INN  ; BLK TOM MELK INN
OUT V0355_UT
; rung 1: V0356
LD SILO_PAST22_0_STATUS  ; Alle objekter som ikke betjenes er ok
LD L3_DREN_PAST22_IND
OR L3_PRODUKT_PAST22_IND  ; INDIVIDADR
ANDLD
AND P22_BLK_TOM_MELK_INN  ; BLK TOM MELK INN
OUT V0356_UT
; rung 2: V0357
LD C15_IND_VST80_K3  ; Z
AND VST80_K3_0_STATUS  ; XX
OUT V0357_UT
; rung 3: V0365
LD SILO_PAST21_0_STATUS  ; Alle objekter som ikke betjenes er ok
LD L4_DREN_PAST21_IND  ; INDIVIDADR
OR L4_PRODUKT_PAST21_IND  ; INDIVIDADR
ANDLD
AND P21_BLK_TOM_MELK_INN  ; BLK TOM MELK INN
OUT V0365_UT
; rung 4: V0366
LD SILO_PAST21_0_STATUS  ; Alle objekter som ikke betjenes er ok
LD L4_DREN_PAST21_IND  ; INDIVIDADR
OR L4_PRODUKT_PAST22_IND  ; INDIVIDADR
ANDLD
AND P22_BLK_TOM_MELK_INN  ; BLK TOM MELK INN
OUT V0366_UT
; rung 5: V2101
LD PGM503_0_STATUS  ; XX
OUT V2101_UT

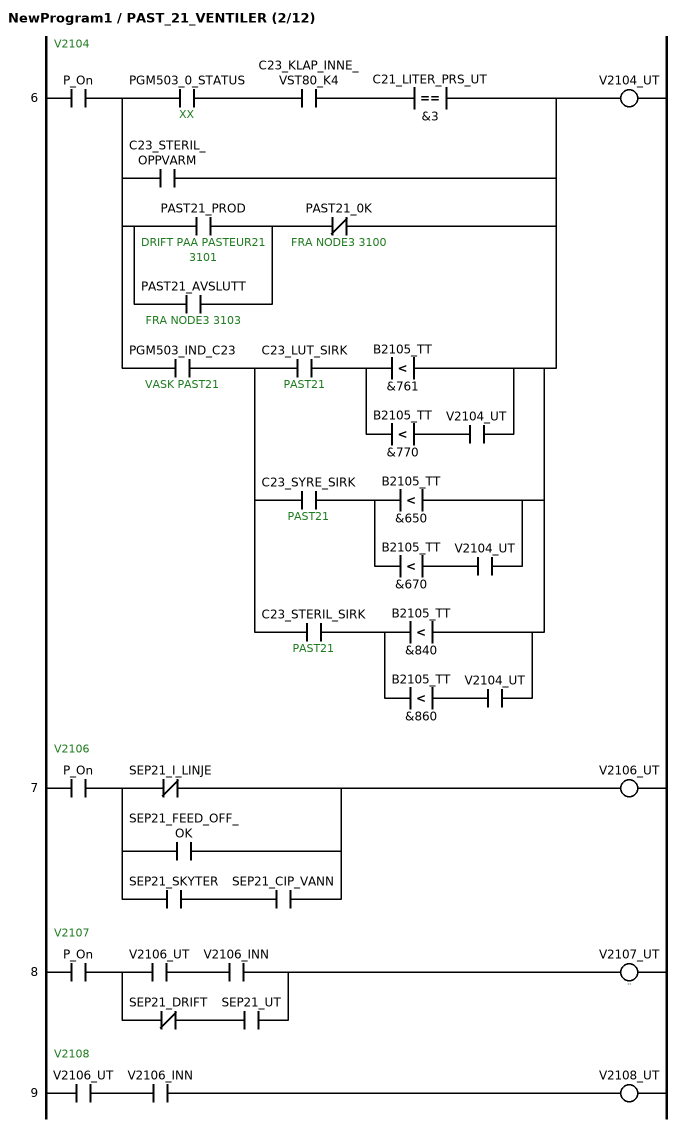
; rung 6: V2104
LD P_On
LD PGM503_0_STATUS  ; XX
AND C23_KLAP_INNE_VST80_K4
AND=(300) C21_LITER_PRS_UT &3
OR C23_STERIL_OPPVARM
LD PAST21_PROD  ; DRIFT PAA PASTEUR21 3101
OR PAST21_AVSLUTT  ; FRA NODE3 3103
ANDNOT PAST21_0K  ; FRA NODE3 3100
ORLD
LD PGM503_IND_C23  ; VASK PAST21
LD C23_LUT_SIRK  ; PAST21
LD<(310) B2105_TT &761
LD<(310) B2105_TT &770
AND V2104_UT
ORLD
ANDLD
LD C23_SYRE_SIRK  ; PAST21
LD<(310) B2105_TT &650
LD<(310) B2105_TT &670
AND V2104_UT
ORLD
ANDLD
ORLD
LD C23_STERIL_SIRK  ; PAST21
LD<(310) B2105_TT &840
LD<(310) B2105_TT &860
AND V2104_UT
ORLD
ANDLD
ORLD
ANDLD
ORLD
ANDLD
OUT V2104_UT
; rung 7: V2106
LD P_On
LDNOT SEP21_I_LINJE
OR SEP21_FEED_OFF_OK
LD SEP21_SKYTER
AND SEP21_CIP_VANN
ORLD
ANDLD
OUT V2106_UT
; rung 8: V2107
LD P_On
LD V2106_UT
AND V2106_INN
LDNOT SEP21_DRIFT
AND SEP21_UT
ORLD
ANDLD
OUT V2107_UT  ; ¨
; rung 9: V2108
LD V2106_UT
AND V2106_INN
OUT V2108_UT

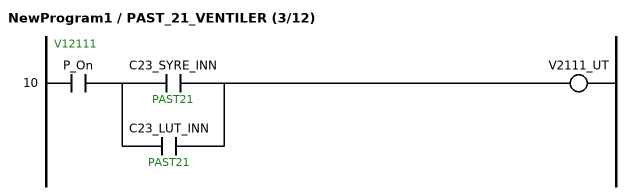
; rung 10: V12111
LD P_On
LD C23_SYRE_INN  ; PAST21
OR C23_LUT_INN  ; PAST21
ANDLD
OUT V2111_UT

